PROGRAM MAIN
VAR
	nState : BYTE;
	fbLinked_List : FB_Linked_List;
	aArray : ARRAY[0..100] OF T_DATA_TYPE;
END_VAR

 CASE nState OF 
	0: // Runs functions once
		fbLinked_List.Init();
		fbLinked_List.Create(1);
		fbLinked_List.Create(2);
		fbLinked_List.Create(3);
		fbLinked_List.Push(12);
		fbLinked_List.Insert(20,2);
		fbLinked_List.Pop();
		
		
		fbLinked_List.Display(aArray);
		nState := nState + 1;
END_CASE

END_PROGRAM

(* stored: Version 1.1.0.1, ProductVersion 3.1.4024.4
   POU MAIN: Id {86dc0999-fc6b-4ce8-a12d-7649401b850c}, SpecialFunc None *)
